PROGRAM MAIN
VAR
	Value1 : INT;
	Value2 : INT;
END_VAR

END_PROGRAM

(* stored: Version 1.1.0.1, ProductVersion 3.1.4022.12
   POU MAIN: Id {5389bffc-5fc7-4629-b6a9-ec8909c13e1e}, SpecialFunc None *)
